FUNCTION_BLOCK FB_SetMode
VAR_INPUT
	bPower : BOOL;
	bOn : BOOL;
	bMode : BOOL;
	bStart : BOOL;
	bStop : BOOL;
END_VAR
VAR_OUTPUT
	eMode : E_Mode;
	sMode : STRING;
	bGreenLight : BOOL;
	bRedLight : BOOL;
END_VAR
VAR
END_VAR



IF bPower = TRUE THEN	
	IF bON = FALSE OR bStart = FALSE OR bStop = TRUE THEN
		eMode		:=	E_Mode.Off;
		bGreenLight	:=	FALSE;
		bRedLight 	:=	TRUE;
	
	ELSIF bON = TRUE AND bStart = TRUE AND bSTOP = FALSE THEN
		IF bMode = FALSE THEN
		eMode := E_Mode.Manual;
		ELSE
		eMode := E_Mode.Auto;
		END_IF
		
	bGreenLight := TRUE;
	bRedLight := FALSE;
		
	END_IF
ELSE
		eMode := E_Mode.Off;
		bGreenLight := FALSE; // No power = No lights
		bRedLight := FALSE;	  // NO power = No lights
END_IF




// String to HMI displaying current mode
IF eMode = E_Mode.Auto THEN
	sMode := 'AUTO';
ELSIF eMode = E_Mode.Manual THEN
	sMode := 'Manual';

ELSE
	sMode := 'OFF';
END_IF

END_FUNCTION_BLOCK

(* stored: Version 1.1.0.1, ProductVersion 3.1.4024.10
   POU FB_SetMode: Id {f209cd25-6b98-40b1-9d47-5c7d8d7039ac}, SpecialFunc None *)
